// TwinCAT 3 PLC project ph_lv1_Communication_Serial
// Title: tclib_ph_lv1_comm_serial
// Company: Poh
// Author: Poh
// ProjectVersion: 0.1.1.0
// ProgramVersion: 3.1.4020.1
// libraries:
//   Tc2_SerialCom, * (Beckhoff Automation GmbH)
//   Tc2_Standard, * (Beckhoff Automation GmbH)
//   Tc2_System, * (Beckhoff Automation GmbH)
//   tclib_ph_lv0, * (Poh)
//   tclib_ph_lv1_generic_communication_interface, * (Poh)
// project tree:
//   Modules/Base Class/ C_SerialBase.TcPOU
//   Modules/ M_EL6_SERIAL.TcPOU, M_PC_SERIAL.TcPOU
// (motion and I/O tree: see PLC project ph_lv0)
// real-time tasks:
//   TASK PlcTask: cycle T#10ms, priority 20, ADS port 350
//   TASK Fast: cycle T#3ms, priority 1, ADS port 351

// ---- Modules/Base Class/C_SerialBase.TcPOU
FUNCTION_BLOCK C_SerialBase IMPLEMENTS IFC_GENERIC_COMMUNICATION_INTERFACE
VAR_INPUT
END_VAR
VAR_OUTPUT
END_VAR
VAR
	//Software Buffers
		_txBuffer : ComBuffer;
		_rxBuffer : ComBuffer;
	//Serial Properties
		_UsePrefix 	: BOOL := FALSE;
		_UseSuffix 	: BOOL := FALSE;
		_Prefix		: STRING(5);
		_Suffix		: STRING(5);
		_LineError	: BOOL := FALSE;
	//Serial FunctionBlocks
		M_RECEIVE	: ReceiveData;
		M_SEND		: SendData;
END_VAR
VAR CONSTANT
	//Read/Write Buffer Size
		_BufferSize : UINT := 300;
END_VAR

METHOD Close_Connection : ph_lv0.RETURN_CODE
Close_Connection := ph_lv0.LV0_RETURNCODE.RETURN_SUCCESS;
END_METHOD

METHOD Create_Handle : ph_lv0.RETURN_CODE
VAR_INPUT
	Configuration	: POINTER TO S_GCI_CONFIG;
	OUT_HANDLE	: POINTER TO UDINT;
END_VAR
Create_Handle := ph_lv0.LV0_RETURNCODE.RETURN_SUCCESS;
END_METHOD

METHOD Open_Connection : ph_lv0.RETURN_CODE
VAR_INPUT
	CONNECTION_INFO	: POINTER TO S_GCI_CONFIG;
END_VAR
IF _LineError THEN
	Open_Connection := ph_lv0.LV0_RETURNCODE.RETURN_ERROR;
ELSE
	Open_Connection := ph_lv0.LV0_RETURNCODE.RETURN_SUCCESS;
END_IF
END_METHOD

PROPERTY Prefix : STRING(5)
GET
Prefix := _Prefix;
END_GET
SET
_Prefix := Prefix;
END_SET
END_PROPERTY

METHOD Read : ph_lv0.RETURN_CODE
VAR_INPUT
	Configuration	: POINTER TO PH_LV1_GENERIC_COMMUNICATION_INTERFACE.S_GCI_CONFIG;
END_VAR
IF _UsePrefix THEN
	M_RECEIVE.pPrefix := ADR(_Prefix);
	M_RECEIVE.LenPrefix := INT_TO_BYTE(LEN(_Prefix));
ELSE
	M_RECEIVE.pPrefix := 0;
	M_RECEIVE.LenPrefix := 0;
END_IF
IF _UseSuffix THEN
	M_RECEIVE.pSuffix := ADR(_Suffix);
	M_RECEIVE.LenSuffix := INT_TO_BYTE(LEN(_Suffix));
ELSE
	M_RECEIVE.pSuffix := 0;
	M_RECEIVE.LenSuffix := 0;
END_IF
M_RECEIVE.Timeout := T#1S;
M_RECEIVE(
	pReceiveData:= Configuration^.P_Data, 
	SizeReceiveData:= Configuration^.Data_Size, 
	RXbuffer:= _rxBuffer);
IF M_RECEIVE.Error <> 0 THEN
	Read := ph_lv0.LV0_RETURNCODE.RETURN_ERROR;
ELSIF NOT _UseSuffix AND M_RECEIVE.RxTimeout THEN
	Read := ph_lv0.LV0_RETURNCODE.RETURN_SUCCESS;
ELSIF M_RECEIVE.DataReceived THEN
	Read := ph_lv0.LV0_RETURNCODE.RETURN_SUCCESS;
ELSE
	Read := ph_lv0.LV0_RETURNCODE.RETURN_BUSY;
END_IF
END_METHOD

METHOD Release_Handle : ph_lv0.RETURN_CODE
VAR_INPUT
	IN_HANDLE	: POINTER TO UDINT;
END_VAR
Release_Handle := ph_lv0.LV0_RETURNCODE.RETURN_SUCCESS;
END_METHOD

PROPERTY Suffix : STRING(5)
GET
Suffix := _Suffix;
END_GET
SET
_Suffix := Suffix;
END_SET
END_PROPERTY

PROPERTY Use_Prefix : BOOL
GET
Use_Prefix := _UsePrefix;
END_GET
SET
_UsePrefix := Use_Prefix;
END_SET
END_PROPERTY

PROPERTY Use_Suffix : BOOL
GET
Use_Suffix := _UseSuffix;
END_GET
SET
_UseSuffix := Use_Suffix;
END_SET
END_PROPERTY

METHOD Write : ph_lv0.RETURN_CODE
VAR_INPUT
	Configuration	: POINTER TO PH_LV1_GENERIC_COMMUNICATION_INTERFACE.S_GCI_CONFIG;
END_VAR
M_SEND(
	pSendData:= Configuration^.P_Data, 
	Length:= Configuration^.Data_Size, 
	Busy=> , 
	Error=> , 
	TXbuffer:= _txBuffer);
IF M_SEND.Error <> 0 THEN
	Write := ph_lv0.LV0_RETURNCODE.RETURN_ERROR;
ELSIF NOT M_SEND.busy THEN
	Write := ph_lv0.LV0_RETURNCODE.RETURN_SUCCESS;
ELSE
	Write := ph_lv0.LV0_RETURNCODE.RETURN_BUSY;
END_IF
END_METHOD

END_FUNCTION_BLOCK

// ---- Modules/M_EL6_SERIAL.TcPOU
FUNCTION_BLOCK M_EL6_SERIAL EXTENDS C_SerialBase
VAR_INPUT
END_VAR
VAR_OUTPUT
END_VAR
VAR
	//Hardware Buffers
		IN_Hardward_Buffer AT %I*	: EL6inData22B;
		OUT_Hardward_Buffer AT %Q*	: EL6outData22B;
		//IN_Hardward_Buffer AT %I*	: PcComInData;
		//OUT_Hardward_Buffer AT %Q* 	: PcComOutData;
	//Serial FunctionBlocks
		M_SERIALCONTROLLER : SerialLineControl;
END_VAR

METHOD Hardware_Buffer_IO : Return_Code
VAR_INPUT
END_VAR
M_SERIALCONTROLLER(
	Mode:= SERIALLINEMODE_EL6_22B, 
	pComIn:= ADR(IN_Hardward_Buffer), 
	pComOut:= ADR(OUT_Hardward_Buffer), 
	SizeComIn:= SIZEOF(IN_Hardward_Buffer), 
	Error=> , 
	ErrorID=> , 
	TxBuffer:= _txBuffer, 
	RxBuffer:= _rxBuffer);
IF M_SERIALCONTROLLER.Error THEN
	_LineError := TRUE;
ELSE
	_LineError := FALSE;
END_IF
END_METHOD

PROPERTY Serial_Line_Error : BOOL
GET
Serial_Line_Error := _LineError;
END_GET
END_PROPERTY

END_FUNCTION_BLOCK

// ---- Modules/M_PC_SERIAL.TcPOU
FUNCTION_BLOCK M_PC_SERIAL Extends C_SerialBase
VAR_INPUT
END_VAR
VAR_OUTPUT
END_VAR
VAR
	//Hardware Buffers
		//IN_Hardward_Buffer AT %I*	: EL6inData22B;
		//OUT_Hardward_Buffer AT %Q*	: EL6outData22B;
		IN_Hardward_Buffer AT %I*	: PcComInData;
		OUT_Hardward_Buffer AT %Q* 	: PcComOutData;
	//Serial FunctionBlocks
		M_SERIALCONTROLLER : SerialLineControl;
END_VAR

METHOD Hardware_Buffer_IO : Return_Code
VAR_INPUT
END_VAR
M_SERIALCONTROLLER(
	Mode:= SERIALLINEMODE_PC_COM_PORT, 
	pComIn:= ADR(IN_Hardward_Buffer), 
	pComOut:= ADR(OUT_Hardward_Buffer), 
	SizeComIn:= SIZEOF(IN_Hardward_Buffer), 
	Error=> , 
	ErrorID=> , 
	TxBuffer:= _txBuffer, 
	RxBuffer:= _rxBuffer);
IF M_SERIALCONTROLLER.Error THEN
	_LineError := TRUE;
ELSE
	_LineError := FALSE;
END_IF
END_METHOD

PROPERTY Serial_Line_Error : BOOL
GET
Serial_Line_Error := _LineError;
END_GET
END_PROPERTY

END_FUNCTION_BLOCK
